// TIA Portal V16 export
// export: Created 2022-11-17T15:49:40.0962394Z, ExportSetting WithDefaults, DisplayName Totally Integrated Automation Portal, DisplayVersion V16 Update 6, DisplayName TIA Portal Version Control Interface, DisplayVersion V16 Update 2, DisplayName TIA Portal Openness, DisplayVersion V16 Update 6, DisplayName SINAMICS Startdrive Advanced, DisplayVersion V16 Update 5, DisplayName SINAMICS Startdrive G130, G150, S120, S150, SINAMICS MV, S210, DisplayVersion V16 Update 5, DisplayName SINAMICS Startdrive G110M, G120, G120C, G120D, G120P, G115D, DisplayVersion V16 Update 5, DisplayName STEP 7 Professional, DisplayVersion V16 Update 6, DisplayName STEP 7 Safety, DisplayVersion V16, DisplayName WinCC Advanced, DisplayVersion V16 Update 6
DATA_BLOCK "DB25_Display"   // DB25
{ S7_Optimized_Access := 'FALSE' }
AUTHOR : Robopac
VERSION : 0.0
// stored: AutoNumber false, IsOnlyStoredInLoadMemory false, IsWriteProtectedInAS false
   VAR RETAIN
      dbw0 : Int := 2;   // Command area 1 (Display Esa)
      dbw2 : Int := 0;   // Command area 2 (Display Esa)
      dbw4 : Int := 0;   // Command area 3 (Display Esa)
      dbw6 : Int := 0;   // Command area 4 (Display Esa)
      dbb8 : Byte := 16#00;   // Status area 1 (Display Esa)
      dbx9_0 : Bool := FALSE;   // Status area 1 (Display Esa): Watchdog
      dbx9_1 : Bool := FALSE;   // Status area 1 (Display Esa): Display in editing
      dbw10 : Int := 0;   // Status area 2 (Display Esa)
      dbw12 : Int := 1;   // Status area 3 Current Page (Display Esa)
      dbw14 : Int := 0;   // Status area 4 (Display Esa)
      dbw16 : Int := 0;
      dbw18 : Int := 2;   // Active program on grey bar
      dbx20_0 : Bool := FALSE;   // Grey bar data 1: Wrapping excluded
      dbx20_1 : Bool := TRUE;   // Grey bar data 1: Wrapping included
      dbx20_2 : Bool := FALSE;   // Grey bar data 1: Wrapping included + Top
      dbx20_3 : Bool := TRUE;   // Grey bar data 1: Pressure plate included/excluded
      dbx20_4 : Bool := FALSE;   // Grey bar data 1: Lifter plate included/excluded
      dbx20_5 : Bool := FALSE;
      dbx20_6 : Bool := FALSE;
      dbx20_7 : Bool := FALSE;
      dbx21_0 : Bool := FALSE;   // Grey bar data 1: Step 1_6 or 7_12(1) shown
      dbx21_1 : Bool := FALSE;   // Grey bar data 1: Data loaded for grey bar
      dbx21_2 : Bool := FALSE;
      dbx21_3 : Bool := FALSE;
      dbx21_4 : Bool := FALSE;
      dbx21_5 : Bool := FALSE;
      dbx21_6 : Bool := FALSE;
      dbx21_7 : Bool := FALSE;
      dbw22 : Int := 5;   // Grey bar data 2: Quote active
      dbw24 : Int := 2;   // Grey bar data 3:
      dbw26 : Int := 0;   // Grey bar data 4:
      dbw28 : Int := 0;   // Grey bar data 5:
      dbw30 : Int := 1;   // Copy of current page
      dbx32_0 : Bool := FALSE;   // Program bit: Load data from data table to display area
      dbx32_1 : Bool := FALSE;   // Program bit: Save data from display area to data table
      dbx32_2 : Bool := FALSE;   // Program bit: Blink load button
      dbx32_3 : Bool := FALSE;   // Program bit: Blink load button
      dbx32_4 : Bool := FALSE;   // Program bit: Blink save button
      dbx32_5 : Bool := FALSE;   // Program bit: Blink save button
      dbx32_6 : Bool := FALSE;   // Program data modified on display
      dbx32_7 : Bool := FALSE;
      dbx33_0 : Bool := FALSE;   // Return to page 1 after 3 minutes
      dbx33_1 : Bool := FALSE;   // Exit from alarm page
      dbx33_2 : Bool := FALSE;   // Support for display communication timeout
      dbx33_3 : Bool := FALSE;   // Jump to no password page
      dbx33_4 : Bool := FALSE;   // Support memory for pressure plate grey bar
      dbx33_5 : Bool := FALSE;   // Support memory for lifter grey bar
      dbx33_6 : Bool := FALSE;   // Display on sysdata or maintenance page
      dbx33_7 : Bool := FALSE;   // Request to reset the counter for wrapped pallet (Micrologix)
      dbw34 : Int := 1;   // Copy of program to be shown on display
      dbw36 : Int := 18;   // Old page used on alarm exit
      dbw38 : Int := 5;   // Support memory for quote active
      dbx40_0 : Bool := FALSE;   // Pallet on conveyor bit: Conveyor CM
      dbx40_1 : Bool := FALSE;   // Pallet on conveyor bit: Conveyor pos.1 (infeed)
      dbx40_2 : Bool := TRUE;   // Pallet on conveyor bit: Conveyor pos.2 (outfeed)
      dbx40_3 : Bool := FALSE;   // Pallet on conveyor bit:
      dbx40_4 : Bool := TRUE;   // Pallet on conveyor bit:
      dbx40_5 : Bool := FALSE;   // Pallet on conveyor bit:
      dbb41 : Byte := 16#00;   // Pallet on rotoplat conveyor byte: 0 empty, 1 pallet, 2 empty 90, 3 pallet 90
      dbw42 : Int := 0;   // Command area 1 (Display Siemens TP) -
      dbw44 : Word := 16#0000;   // Command area 2 (Display Siemens TP)
      dbw46 : Word := 16#0000;   // Command area 3 (Display Siemens TP)
      dbw48 : Word := 16#0000;   // Command area 4 (Display Siemens TP)
      dbb50 : Byte := 16#00;   // Status area (Display Siemens TP):
      dbx51_0 : Bool := TRUE;   // Status area (Display Siemens TP): Start bit
      dbx51_1 : Bool := FALSE;   // Status area (Display Siemens TP): Display offline/online
      dbx51_2 : Bool := FALSE;   // Status area (Display Siemens TP): Watchdog
      dbw52 : Word := 16#0001;   // Status area (Display Siemens TP): Current page type
      dbw54 : Int := 1;   // Status area (Display Siemens TP): Current page number
      dbw56 : Word := 16#0000;   // Status area (Display Siemens TP): Reserved
      dbw58 : Word := 16#0001;   // Status area (Display Siemens TP): Current object number
      dbw60 : Word := 16#0000;   // Status area (Display Siemens TP): Reserved
      ProgQuoteQX : Int := 0;   // Multiplex Wincc - Program data
      ProgBitQX : Int := 4;   // Multiplex Wincc - Program data
      ProgQuotaQX : Int := 2;   // Multiplex Wincc - Program data
      ProgGiriQX : Int := 6;   // Multiplex Wincc - Program data
      ProgSovrappQX : Int := 0;   // Multiplex Wincc - Program data
      ProgStringifasciaQX : Int := 8;   // Multiplex Wincc - Program data
      ProgTiroFilmQX : Int := 10;   // Multiplex Wincc - Program data
      ProgPrestiroFilmQX : Int := 12;   // Multiplex Wincc - Program data
      ProgStringifascia2QX : Int := 9;   // Multiplex Wincc - Program data
      dbw80 : Int := 3;   // Multiplex Wincc - Program data
      dbw82 : Int := 0;
      dbw84 : Int := 0;
      dbw86 : Int := 0;
      dbw88 : Int := 0;
      dbw90 : Int := 0;
      dbw92 : Int := 0;
      dbw94 : Int := 0;
      dbw96 : Int := 0;
      dbw98 : Int := 130;
   END_VAR
BEGIN
END_DATA_BLOCK
